(* PLC project Skill-Test-Projekt.project, CODESYS CODESYS V3.5 SP16 Patch 1 *)
(* stored: creationDateTime 2022-10-13T18:01:38.0272131, modificationDateTime 2022-10-12T10:05:12.0722967 *)

PROGRAM PLC_PRG
  VAR
    drillingSkill_1 : DrillingSkill;
    punchingSkill_1 : PunchingSkill;
  END_VAR

                    drillingSkill_1();
punchingSkill_1();

                  
END_PROGRAM

FUNCTION_BLOCK DrillingSkill EXTENDS PLC2Skill.Skill
  VAR_INPUT
    numberOfHoles : PLC2Skill.SkillParameter := (default := 10, name := 'numberOfHoles', paramType := 'int', required := TRUE);
  END_VAR
  VAR_OUTPUT
    drillingResult : PLC2Skill.SkillParameter := (default := 0, name := 'drillingResult', paramType := 'bool', required := TRUE);
  END_VAR

                    
                  

METHOD execute : BOOL
                          THIS^.drillingResult.value := TO_INT(true);
                        
END_METHOD

METHOD resetting : BOOL
                          THIS^.drillingResult.value := TO_INT(false);
                        
END_METHOD
END_FUNCTION_BLOCK

FUNCTION_BLOCK PunchingSkill EXTENDS PLC2Skill.Skill
  VAR_INPUT
    numberOfHoles : PLC2Skill.SkillParameter := (default := 10, name := 'numberOfHoles', paramType := 'int', required := TRUE);
  END_VAR
  VAR_OUTPUT
    drillingResult : PLC2Skill.SkillParameter := (default := 0, name := 'drillingResult', paramType := 'bool', required := TRUE);
  END_VAR

                    
                  

METHOD execute : BOOL
                          THIS^.drillingResult.value := TO_INT(true);
                        
END_METHOD

METHOD resetting : BOOL
                          THIS^.drillingResult.value := TO_INT(false);
                        
END_METHOD
END_FUNCTION_BLOCK

CONFIGURATION Device
  RESOURCE Application ON PLC
    TASK MainTask(INTERVAL := T#20ms, PRIORITY := 1);
    PROGRAM PLC_PRG WITH MainTask : PLC_PRG;
  END_RESOURCE
END_CONFIGURATION
